Staubli VAL3: getTool.pgx

public program getTool(num& x_nTool)
begin
  //
  // get the tool
  //
  x_nTool=jEditPoint.nIndexTool
end
